// TwinCAT 3 PLC project Untitled1
// ProgramVersion: 3.1.4024.0
// libraries:
//   Tc2_Standard, * (Beckhoff Automation GmbH)
//   Tc2_System, * (Beckhoff Automation GmbH)
//   Tc3_JsonXml, * (Beckhoff Automation GmbH)
//   Tc3_Module, * (Beckhoff Automation GmbH)
// project tree:
//   / PlcTask.TcTTO
//   POUs/ FB_ReadJsonReal.TcPOU, FB_SaveFile.TcPOU, MAIN.TcPOU
// real-time tasks:
//   TASK PlcTask: cycle T#10ms, priority 20, ADS port 350

CONFIGURATION Untitled1
    RESOURCE PLC ON TwinCAT3
        TASK PlcTask(INTERVAL := T#10ms, PRIORITY := 20);
        PROGRAM MAIN WITH PlcTask : MAIN;
    END_RESOURCE
END_CONFIGURATION

// ---- POUs/MAIN.TcPOU
PROGRAM MAIN
VAR
	fbJson:FB_JsonSaxWriter;
	fbJsonDomParser:FB_JsonDomParser;

	fbSaveFile :FB_SaveFile;
	fbReadJsonReal :FB_ReadJsonReal;
	
	jsonDOC : SJsonValue;
	
	Trigger: BOOL:=TRUE;
	sBuffer :STRING(100);
	r32:REAL;

	bSave:BOOL;

	
	bLoadJsonFile:BOOL;
	jSonProp :SJsonValue;
	jsonRoot :SJsonValue;
	fSensorValue :LREAL;
	bReadValue:BOOL;
END_VAR


IF Trigger THEN
	r32:=r32+0.01;
	IF r32>=1000.0 THEN
		r32:=0.0;
	END_IF

	//Object creation
	fbJson.StartObject(); //Open Bracket
		fbJson.AddKey('Sensor1');
		fbJson.AddReal((r32));
	fbJson.EndObject(); //Close Bracket
	
	//Document creation
	sBuffer := fbJson.GetDocument();
	fbJson.ResetDocument();
	
END_IF

//Save information
IF bSave THEN
	fbSaveFile(sPath:='C:\TwinCAT\3.1\Boot\MyData.json',AmsNetId:='',sBuffer:=sBuffer);
	bSave:=FALSE;
END_IF

//Read information
IF bLoadJsonFile THEN
fbReadJsonReal(Member:='Sensor1',sPath:='C:\TwinCAT\3.1\Boot\MyData.json',fReadValue=>);
fSensorValue:= fbReadJsonReal.fReadValue;
END_IF

END_PROGRAM

// ---- POUs/FB_SaveFile.TcPOU
FUNCTION_BLOCK FB_SaveFile
VAR_INPUT
	sPath:STRING;
	AmsNetId:STRING;
	sBuffer:STRING;
END_VAR
VAR_OUTPUT
END_VAR
VAR
	//Functions
	fbFileOpen   : FB_FileOpen;
    fbFileWrite  : FB_FileWrite;
    fbFileClose  : FB_FileClose;

	//Aux variables
	jsonDOC : SJsonValue;
	FileHandle :UINT;
	nState: INT:=0;
	
	bOpenExec:BOOL;
	bWriteExec:BOOL;
	bCloseExec:BOOL;
	
	nErrorIdOpen:UDINT;
	nErrorIdWrite:UDINT;
	nErrorIdClose:UDINT;
END_VAR

CASE nState OF
	00: //Idle
	bOpenExec:=FALSE;
	bWriteExec:=FALSE;
	bCloseExec:=FALSE;
	nState:=10;
		
	
	10://CreateFile
		bOpenExec:=TRUE;
		fbFileOpen(sNetId:=AmsNetId,sPathName := sPath,nMode := FOPEN_MODEWRITE OR FOPEN_MODETEXT,bExecute := bOpenExec);
		FileHandle :=fbFileOpen.hFile;
		IF NOT fbFileOpen.bError AND NOT fbFileOpen.bBusy THEN
		nState:=20;
		bOpenExec := FALSE;
		END_IF
		IF fbFileOpen.bError THEN
		nState :=999;			
		END_IF
		
	20: //Write the information
		bWriteExec:=TRUE;
		fbFileWrite(sNetId := '',hFile := FileHandle,pWriteBuff := ADR(sBuffer),cbWriteLen := LEN(sBuffer),bExecute := bWriteExec);
		IF NOT fbFileWrite.bError AND NOT fbFileWrite.bBusy THEN
		bWriteExec :=FALSE;
		nState :=30;
		END_IF
		IF fbFileWrite.bError THEN
		nState :=999;			
		END_IF
		
	30: //Save the information and close the file
		bCloseExec:=TRUE;
		fbFileClose(sNetId:='', hFile := FileHandle, bExecute := bCloseExec);
		IF NOT fbFileClose.bError AND NOT fbFileClose.bBusy THEN
		FileHandle:=0;
		bCloseExec := FALSE;
		END_IF
		IF fbFileClose.bError THEN
		nState :=999;			
		END_IF
		
	999: //Error State
		nErrorIdOpen:=fbFileOpen.nErrId;
		nErrorIdWrite:=fbFileWrite.nErrId;
		nErrorIdClose:=fbFileClose.nErrId;	
	END_CASE

END_FUNCTION_BLOCK

// ---- POUs/FB_ReadJsonReal.TcPOU
FUNCTION_BLOCK FB_ReadJsonReal
VAR_INPUT
	Member:STRING;
	sPath:STRING;
END_VAR
VAR_OUTPUT
	fReadValue:LREAL;
END_VAR
VAR
	nState: INT:=0;
	fbJsonDomParser:FB_JsonDomParser;
	ErrorCode :HRESULT;
	jSonProp :SJsonValue;
	jsonRoot :SJsonValue;
	bLoadDocument:BOOL;
END_VAR


CASE nState OF
	00: //Idle
		bLoadDocument:=FALSE;
		nState:=10;
		
	10: //Load the document
		bLoadDocument:=TRUE;
		fbJsonDomParser.LoadDocumentFromFile(sPath,bLoadDocument, hrErrorCode =>ErrorCode);
		IF ErrorCode = S_OK THEN
		nState:=20;
		END_IF
	
	20: //Read the desired values
		jsonRoot :=fbJsonDomParser.GetDocumentRoot();
		jSonProp := fbJsonDomParser.FindMember(jsonRoot,Member);
		IF (jsonProp<>0) THEN
			fReadValue := fbJsonDomParser.GetDouble(jSonProp);
		ELSE 
			fReadValue := -999999;
		END_IF
		
END_CASE

END_FUNCTION_BLOCK
